FUNCTION_BLOCK fbMotorisedCB
VAR_INPUT
END_VAR
VAR_OUTPUT
END_VAR
VAR
END_VAR
VAR_IN_OUT
	
END_VAR

END_FUNCTION_BLOCK

(* stored: Version 1.1.0.1, ProductVersion 3.1.4024.11
   POU fbMotorisedCB: Id {0694e418-c73d-46ac-9391-384815d288cb}, SpecialFunc None *)
